// SIMATIC S7-200 project (STEP 7-Micro/WIN), CPU 224 REL 02.01

SYMBOL_TABLE USUARIO1
P_MARCHA         I0.0
C_FOTOELECTRICA  I0.1
P_PARO           I0.2
LED_PARO         Q0.0
LED_MARCHA       Q0.1
C_TRANSPORTADORA Q0.2
P_EXPANDIDO      Q0.3
P_CONTRAIDO      Q0.4
CONTADOR         VW4
END_SYMBOL_TABLE

SYMBOL_TABLE Símbolos S7-200
Primer_ciclo_ON  SM0.1    // ON sólo en el primer ciclo
END_SYMBOL_TABLE

ORGANIZATION_BLOCK PRINCIPAL:OB1
TITLE=COMENTARIOS DEL PROGRAMA
BEGIN
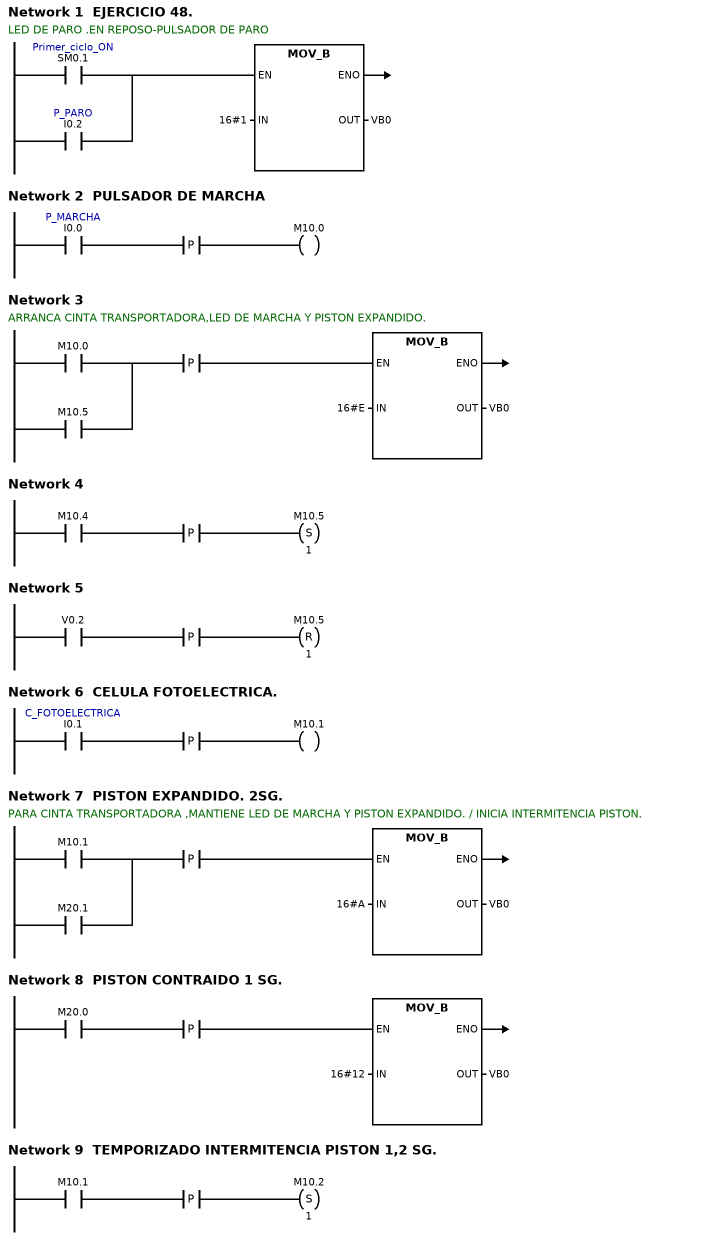
Network 1 // EJERCICIO 48.
// LED DE PARO .EN REPOSO-PULSADOR DE PARO
LD     Primer_ciclo_ON:SM0.1
O      P_PARO:I0.2
MOVB   16#1, VB0
Network 2 // PULSADOR DE MARCHA
LD     P_MARCHA:I0.0
EU
=      M10.0
Network 3
// ARRANCA CINTA TRANSPORTADORA,LED DE MARCHA Y PISTON EXPANDIDO.
LD     M10.0
O      M10.5
EU
MOVB   16#E, VB0
Network 4
LD     M10.4
EU
S      M10.5, 1
Network 5
// (network saved uncompiled; LAD cells follow)
// row 0: c0 -| |- V0.2  c1 -|P|-  c2 -(R) M10.5, 1
Network 6 // CELULA FOTOELECTRICA.
LD     C_FOTOELECTRICA:I0.1
EU
=      M10.1
Network 7 // PISTON EXPANDIDO. 2SG.
// PARA CINTA TRANSPORTADORA ,MANTIENE LED DE MARCHA Y PISTON EXPANDIDO.
// INICIA INTERMITENCIA PISTON.
LD     M10.1
O      M20.1
EU
MOVB   16#A, VB0
Network 8 // PISTON CONTRAIDO 1 SG.
LD     M20.0
EU
MOVB   16#12, VB0
Network 9 // TEMPORIZADO INTERMITENCIA PISTON 1,2 SG.
LD     M10.1
EU
S      M10.2, 1
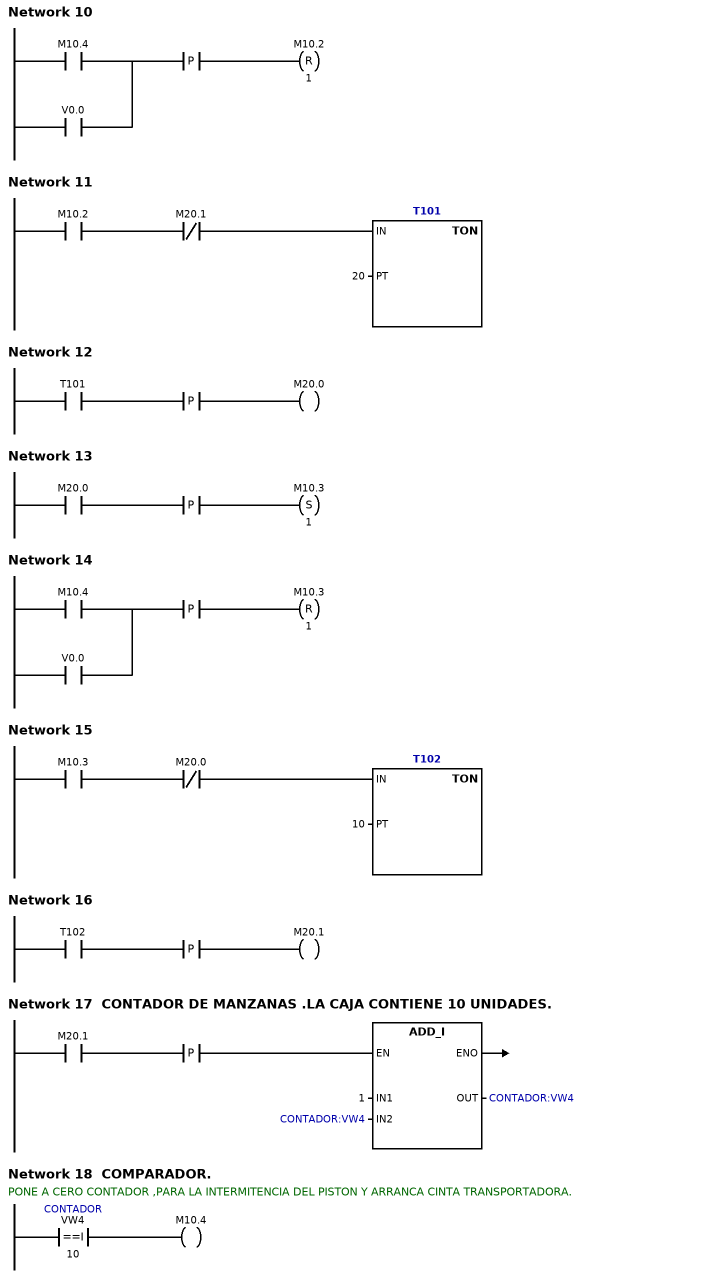
Network 10
// (network saved uncompiled; LAD cells follow)
// row 0: c0 -| |- M10.4 v  c1 -|P|-  c2 -(R) M10.2, 1
// row 1: c0 -| |- V0.0 ^
Network 11
LD     M10.2
AN     M20.1
TON    T101, 20
Network 12
LD     T101
EU
=      M20.0
Network 13
LD     M20.0
EU
S      M10.3, 1
Network 14
// (network saved uncompiled; LAD cells follow)
// row 0: c0 -| |- M10.4 v  c1 -|P|-  c2 -(R) M10.3, 1
// row 1: c0 -| |- V0.0 ^
Network 15
LD     M10.3
AN     M20.0
TON    T102, 10
Network 16
LD     T102
EU
=      M20.1
Network 17 // CONTADOR DE MANZANAS .LA CAJA CONTIENE 10 UNIDADES.
LD     M20.1
EU
+I     1, CONTADOR:VW4
Network 18 // COMPARADOR.
// PONE A CERO CONTADOR ,PARA LA INTERMITENCIA DEL PISTON Y ARRANCA CINTA TRANSPORTADORA.
LDW=   CONTADOR:VW4, 10
=      M10.4
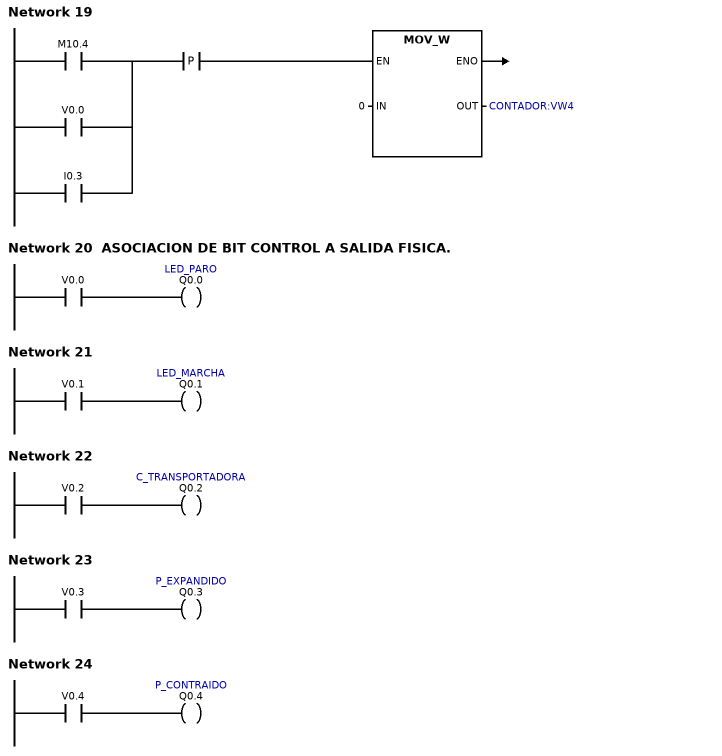
Network 19
// (network saved uncompiled; LAD cells follow)
// row 0: c0 -| |- M10.4 v  c1 -|P|-  c2 --  c3 [MOV_W EN:=power@row0, IN:=0, ENO=>power, OUT=>CONTADOR:VW4]  c4 ->
// row 1: c0 -| |- V0.0 ^v  c3 [box]
// row 2: c0 -| |- I0.3 ^
Network 20 // ASOCIACION DE BIT CONTROL A SALIDA FISICA.
LD     V0.0
=      LED_PARO:Q0.0
Network 21
LD     V0.1
=      LED_MARCHA:Q0.1
Network 22
LD     V0.2
=      C_TRANSPORTADORA:Q0.2
Network 23
LD     V0.3
=      P_EXPANDIDO:Q0.3
Network 24
LD     V0.4
=      P_CONTRAIDO:Q0.4
END_ORGANIZATION_BLOCK
